(*
SPDX-FileCopyrightText: © 2026 Oleksandr Tiutyk <trofimich@gmail.com>
SPDX-License-Identifier: MIT
License: https://opensource.org/license/mit
*)

{attribute 'qualified_only'}
VAR_GLOBAL
	CodeExecutionPhase : BOOL;
	CycleCounter : LWORD;
END_VAR

(* stored: Version 1.1.0.1
   GVL GlobalState: Id {5704066d-1f24-45f5-ae23-8ef26a6bb50a} *)
